PROGRAM MAIN
VAR
	ENCODER : AXIS_REF;
	MOTOR	: AXIS_REF;
END_VAR

END_PROGRAM

(* stored: Version 1.1.0.1, ProductVersion 3.1.4024.14
   POU MAIN: Id {a7a322e6-ffe6-458a-a0c6-07c7acc5ec11}, SpecialFunc None *)
